// TIA Portal V19 export
FUNCTION_BLOCK "CallInterfaceSignals"   // FB38, LAD
TITLE = CallInterfaceSignals
AUTHOR : Siemens Digital Industry
VERSION : 1.0
// The block serves as a calling interface of the block “LAF_InterfaceSignalsBool“. The block is designed as function block in order to implement the block calls as multi-instances.
// Der Baustein dient als Aufrufschnittstelle für den Funktionsbaustein „LSicar_InterfaceSignalsBool“. Er ist als Funktionsbaustein ausgeführt, um die intern aufgerufenen FBs mittels Multiinstanzen realisieren zu können.  
// Die Funktionsbausteine und das zugehörige WinCC-Bild sind für 16 Signaldatensätze („Schnittstelle Signale 01“ … „Schnittstellen Signale 16“) mit jeweils 32 boolschen Signalen vorgesehen.  
// 
// **PLC-Datentypen**  
//  LSicar_typeInterfaceSignalsBool 
//  typeInterfaceSignalsHmi 
//  LSicar _typeInterfaceSignals 
// 
// **WinCC-Diagnosebild**  
// 
// ![Icon](_Icon/reference.PNG)
// 
// siehe ..\Library Types\LSicar_InterfaceSignalsBool.pdf  
// 
//  
// 
// **Beispielaufruf**  
// Abbildung in Kontaktplan (KOP).  D:\Software\Symbols_Icons\BMPs-JPGs-PNGs\Verschiedene\symb_user_goto_transparent.pngEin lauffähiger Programm-Aufruf hierzu ist im „SICAR-StartUp“-Projekt enthalten.  
// 
// **Aufrufschnittstelle**  
// Der Baustein wird einmalig im zyklischen Programm aufgerufen.  
// 
// **Intern verwendete „Erweiterte Anweisungen / Bausteine“**  
// ..\Library Types\LSicar_InterfaceSignalsBool.pdf
// stored: IsIECCheckEnabled true, MemoryReserve 100, SetENOAutomatically true
   VAR
      statReadValueHmi : Bool;   // HMI: Lese Signalwert / HMI: Read value signal
      statSelectSignalsHmi : USInt := 1;   // HMI: Angewählte Interface Schnittstelle (1..16) / HMI: Selected interface signals (1..16)
      statSelectSignalsOld { ExternalAccessible := 'False'; ExternalVisible := 'False'; ExternalWritable := 'False'} : USInt;   // Altwert: Angewählte Interface Schnittstelle / Old value: Selected interface signals
      statRisEdgeReadName { ExternalAccessible := 'False'; ExternalVisible := 'False'; ExternalWritable := 'False'} : Bool;   // Steigende Flanke / Rising edge
      statPosPulseReadName : Bool;   // Positiver Impuls / Positive pulse
      statInterfaceSignalsHmi : Array[0..16] of "LAF_typeInterfaceSignalsHmi";   // HMI: Beschreibung, Wert und Symbolischer Name / HMI: Description, value and symbolic name
      instSignals1Left { S7_SetPoint := 'True'} : "LAF_InterfaceSignalsBool";
      instSignals1Right { ExternalAccessible := 'False'; ExternalVisible := 'False'; ExternalWritable := 'False'} : "LAF_InterfaceSignalsBool";   // Schnittstellen Signale Bild 1 rechts / interface signals screen 1 right
      instSignals2Left { ExternalAccessible := 'False'; ExternalVisible := 'False'; ExternalWritable := 'False'} : "LAF_InterfaceSignalsBool";   // Schnittstellen Signale Bild 2 links / interface signals screen 2 left
      instSignals2Right { ExternalAccessible := 'False'; ExternalVisible := 'False'; ExternalWritable := 'False'} : "LAF_InterfaceSignalsBool";   // Schnittstellen Signale Bild 2 rechts / interface signals screen 2 right
      instSignals3Left { ExternalAccessible := 'False'; ExternalVisible := 'False'; ExternalWritable := 'False'} : "LAF_InterfaceSignalsBool";   // Schnittstellen Signale Bild 3 links / interface signals screen 3 left
      instSignals3Right { ExternalAccessible := 'False'; ExternalVisible := 'False'; ExternalWritable := 'False'} : "LAF_InterfaceSignalsBool";   // Schnittstellen Signale Bild 3 rechts / interface signals screen 3 right
      instSignals4Left { ExternalAccessible := 'False'; ExternalVisible := 'False'; ExternalWritable := 'False'} : "LAF_InterfaceSignalsBool";   // Schnittstellen Signale Bild 4 links / interface signals screen 4 left
      instSignals4Right { ExternalAccessible := 'False'; ExternalVisible := 'False'; ExternalWritable := 'False'} : "LAF_InterfaceSignalsBool";   // Schnittstellen Signale Bild 4 rechts / interface signals screen 4 right
      instSignals5Left { ExternalAccessible := 'False'; ExternalVisible := 'False'; ExternalWritable := 'False'} : "LAF_InterfaceSignalsBool";   // Schnittstellen Signale Bild 5 links / interface signals screen 5 left
      instSignals5Right { ExternalAccessible := 'False'; ExternalVisible := 'False'; ExternalWritable := 'False'} : "LAF_InterfaceSignalsBool";   // interface signals screen 5 right / Schnittstellen Signale Bild 5 rechts
   END_VAR
   VAR_TEMP
      tempLoopCounter : DInt;   // temp. Schleifenzähler / temp. Loop Counter
   END_VAR
   VAR_TEMP   // added for the SCL form of the ladder/FBD networks
      _w1 : Bool;
   END_VAR
BEGIN

REGION Network 1: BLOCK INFO HEADER / Beschreibung
   // SIEMENS AG / (c)Copyright 2024
   // ------------------------------------------------------------------------------
   // Title:            CallInterfaceSignals (FB38)
   // Comment/Function: The block serves as a calling interface of the block “LAF_InterfaceSignalsBool“. The block is designed as function block in order to implement the block calls as multi-instances. 
   // Library/Family:   -
   // Author:           Siemens Digital Industry
   // Tested with:      ---
   // Engineering:      TIA Portal V19
   // Restrictions:     -
   // Requirements:     ---
   // ------------------------------------------------------------------------------
   // Change log table:
   // Version  | Date       | Expert in charge       | Changes applied
   // ---------|------------|------------------------|------------------------------
   // 01.00.00 | 11.12.2023 | SIMATIC Systems Support 
   //                         First released version
   // **Betriebsart Automatik / Hand**  
   // Der Baustein ist keiner Betriebsart / Betriebsartenbereich zugeordnet.  
   // 
   // **Alarme**  
   // Der Baustein generiert keine Alarme.  
   // 
   // #### PLC-Datentypen  
   // Verwendete PLC-Datentypen für den SPS-Programmbaustein und das zugehörige WinCC-Bild.  
   // 
   // {.pageWidth}
   // ![Image](CallInterfaceSignals/de/image1.PNG)
   //  
   //  
   // #### Bausteinaufrufe 
   // Der Baustein “LSicar_InterfaceSignalsBool“ wird in diesem FB als Multi-Instanz aufgerufen, entspr. nebenstehender beispielhafter Darstellung.  
   // 
   // {.pageWidth}
   // ![Image](CallInterfaceSignals/de/image2.PNG)
   //  
   // Um einen neuen FB aufzurufen, ziehen Sie den FB in ein neues Netzwerk, wählen Sie „Multiinstanz“ aus, vergeben Sie einen Namen und parametrieren Sie den FB-Aufruf.  
   // 
   // {.pageWidth}
   // ![Image](CallInterfaceSignals/de/image3.PNG)
   //  
   //  
   // #### Weitere Hinweise 
   // 
   // #### Updateinfo 
   // 
   // #### Weitere Dokumente 
   // 
   // ![Icon](_Icon/reference.PNG)
   // 
   // ..\Library Types\LSicar_InterfaceSignalsBool.pdf
END_REGION

REGION Network 2: DESCRIPTION
   // Function block and corresponding WinCC screen are prepared for 16 data sets (“InterfaceSignals01“ through .”InterfaceSignals16“) with 32 Boolean signals each.  
   // 
   // **PLC-Data types**   
   // 
   // * LAF_typeInterfaceSignalsBool 
   // * LAF _typeInterfaceSignals 
   // * typeInterfaceSignalsHmi 
   // 
   // **WinCC-Faceplate**  
   // 
   // <None> 
   // 
   // **WinCC Diagnostic screen**   
   // 
   // See: ..\Library Types\LAF_InterfaceSignalsBool.pdf  
   // 
   // **Block call example** 
   // 
   // View in ladder-logic (LAD), without parameter settings.  
   // 
   // 
   // **Calling interface**  
   // 
   // The block is be called once in the cyclic program.  
   // 
   // **Internally used „Extended instructions / blocks“**  
   // 
   // See: ..\Library Types\LAF_InterfaceSignalsBool.pdf
END_REGION

REGION Network 3: Initialization Loop_1 / Initialisierung Loop_1
   // Preset the loop index / Vorbesetzen des Schleifenindex
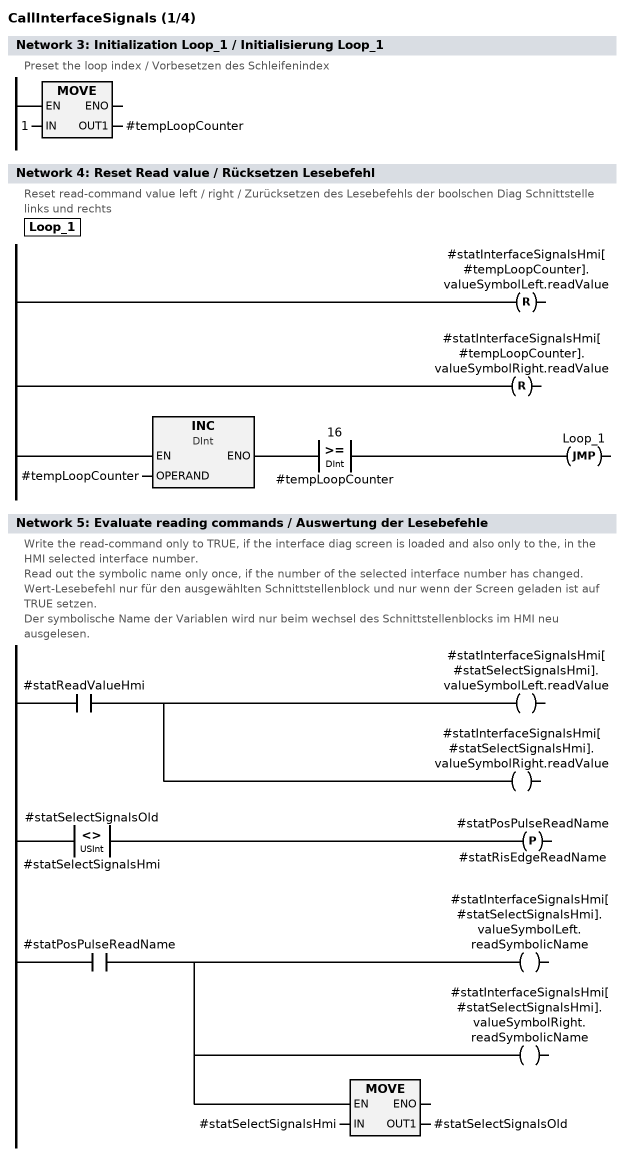
   RUNG wire#powerrail
      Move(in := 1, out1 => #tempLoopCounter)
   END_RUNG
   // the same network as SCL:
   #tempLoopCounter := 1;
END_REGION

REGION Network 4: Reset Read value / Rücksetzen Lesebefehl
   // Reset read-command value left / right / Zurücksetzen des Lesebefehls der boolschen Diag Schnittstelle links und rechts
   Label( Loop_1 )
   RUNG wire#powerrail
      R_Coil( #statInterfaceSignalsHmi[#tempLoopCounter].valueSymbolLeft.readValue )
   END_RUNG
   RUNG wire#powerrail
      R_Coil( #statInterfaceSignalsHmi[#tempLoopCounter].valueSymbolRight.readValue )
   END_RUNG
   RUNG wire#powerrail
      { S7_Templates := "DestType := DInt" } Inc( #tempLoopCounter )
      { S7_Templates := "SrcType := DInt" } GE_Contact(in1 := 16, in2 := #tempLoopCounter)
      JumpCoil( Loop_1 )
   END_RUNG
   // the same network as SCL:
   Loop_1:
   #statInterfaceSignalsHmi[#tempLoopCounter].valueSymbolLeft.readValue := FALSE;
   #statInterfaceSignalsHmi[#tempLoopCounter].valueSymbolRight.readValue := FALSE;
   #tempLoopCounter := #tempLoopCounter + 1;
   IF 16 >= #tempLoopCounter THEN GOTO Loop_1; END_IF;
END_REGION

REGION Network 5: Evaluate reading commands / Auswertung der Lesebefehle
   // Write the read-command only to TRUE, if the interface diag screen is loaded and also only to the, in the HMI selected interface number.
   // Read out the symbolic name only once, if the number of the selected interface number has changed.
   // Wert-Lesebefehl nur für den ausgewählten Schnittstellenblock und nur wenn der Screen geladen ist auf TRUE setzen.
   // Der symbolische Name der Variablen wird nur beim wechsel des Schnittstellenblocks im HMI neu ausgelesen.
   #statInterfaceSignalsHmi[#statSelectSignalsHmi].valueSymbolLeft.readValue := #statReadValueHmi;
   #statInterfaceSignalsHmi[#statSelectSignalsHmi].valueSymbolRight.readValue := #statReadValueHmi;
   #_w1 := #statSelectSignalsOld <> #statSelectSignalsHmi;
   #statPosPulseReadName := #_w1 AND NOT #statRisEdgeReadName;   // rising edge
   #statRisEdgeReadName := #_w1;
   #statInterfaceSignalsHmi[#statSelectSignalsHmi].valueSymbolLeft.readSymbolicName := #statPosPulseReadName;
   #statInterfaceSignalsHmi[#statSelectSignalsHmi].valueSymbolRight.readSymbolicName := #statPosPulseReadName;
   IF #statPosPulseReadName THEN #statSelectSignalsOld := #statSelectSignalsHmi; END_IF;
END_REGION

REGION Network 6: Interface Signals 01 / Interface Signals 01 -Example: Model PosDev+Lifter - IN/OUT-
   // Aufruf des Schnittstellen Signal Bausteins Ba-Bereich 1
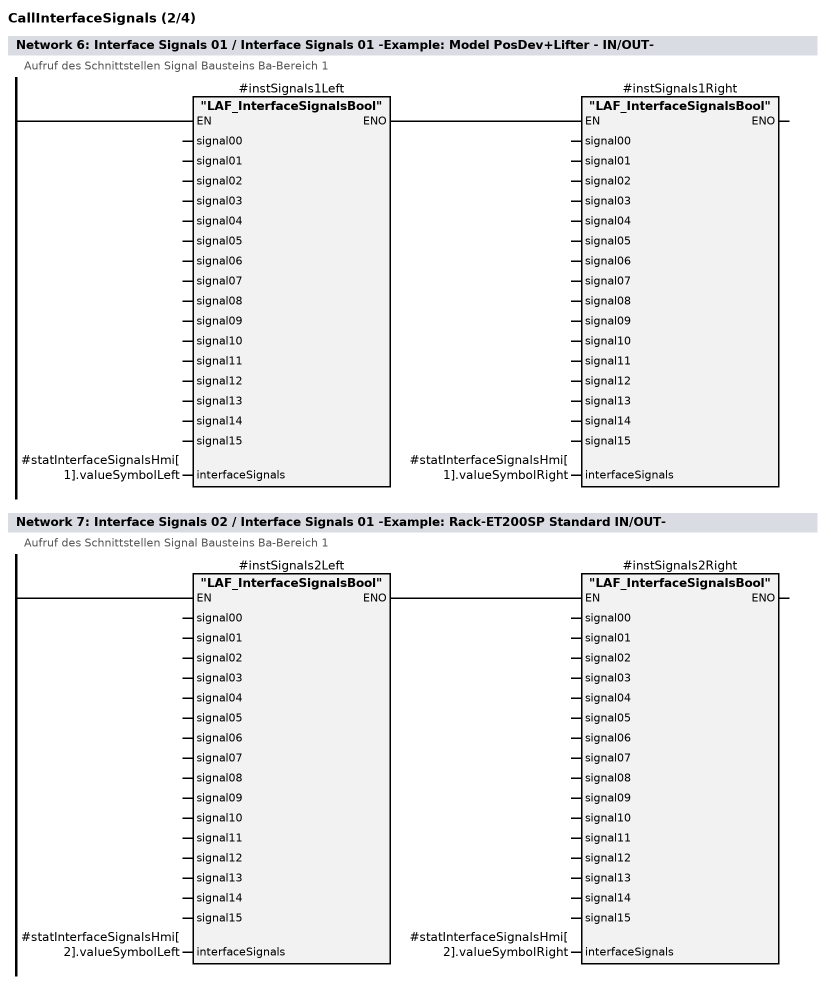
   RUNG wire#powerrail
      #instSignals1Left(signal00 :=, signal01 :=, signal02 :=, signal03 :=, signal04 :=, signal05 :=, signal06 :=, signal07 :=, signal08 :=, signal09 :=, signal10 :=, signal11 :=, signal12 :=, signal13 :=, signal14 :=, signal15 :=, interfaceSignals := #statInterfaceSignalsHmi[1].valueSymbolLeft)
      #instSignals1Right(signal00 :=, signal01 :=, signal02 :=, signal03 :=, signal04 :=, signal05 :=, signal06 :=, signal07 :=, signal08 :=, signal09 :=, signal10 :=, signal11 :=, signal12 :=, signal13 :=, signal14 :=, signal15 :=, interfaceSignals := #statInterfaceSignalsHmi[1].valueSymbolRight)
   END_RUNG
   // the same network as SCL:
   #instSignals1Left(interfaceSignals := #statInterfaceSignalsHmi[1].valueSymbolLeft, ENO => #_w1);   // "LAF_InterfaceSignalsBool"
   IF #_w1 THEN
       #instSignals1Right(interfaceSignals := #statInterfaceSignalsHmi[1].valueSymbolRight);   // "LAF_InterfaceSignalsBool"
   END_IF;
END_REGION

REGION Network 7: Interface Signals 02 / Interface Signals 01 -Example: Rack-ET200SP Standard IN/OUT-
   // Aufruf des Schnittstellen Signal Bausteins Ba-Bereich 1
   RUNG wire#powerrail
      #instSignals2Left(signal00 :=, signal01 :=, signal02 :=, signal03 :=, signal04 :=, signal05 :=, signal06 :=, signal07 :=, signal08 :=, signal09 :=, signal10 :=, signal11 :=, signal12 :=, signal13 :=, signal14 :=, signal15 :=, interfaceSignals := #statInterfaceSignalsHmi[2].valueSymbolLeft)
      #instSignals2Right(signal00 :=, signal01 :=, signal02 :=, signal03 :=, signal04 :=, signal05 :=, signal06 :=, signal07 :=, signal08 :=, signal09 :=, signal10 :=, signal11 :=, signal12 :=, signal13 :=, signal14 :=, signal15 :=, interfaceSignals := #statInterfaceSignalsHmi[2].valueSymbolRight)
   END_RUNG
   // the same network as SCL:
   #instSignals2Left(interfaceSignals := #statInterfaceSignalsHmi[2].valueSymbolLeft, ENO => #_w1);   // "LAF_InterfaceSignalsBool"
   IF #_w1 THEN
       #instSignals2Right(interfaceSignals := #statInterfaceSignalsHmi[2].valueSymbolRight);   // "LAF_InterfaceSignalsBool"
   END_IF;
END_REGION

REGION Network 8: Interface Signals 03 / Interface Signals 03 -Example: System flags & Clock flags-
   // Call the interface signals bool blocks of system tags / Aufruf des Schnittstellen Signal Bausteins für die Systemvariablen
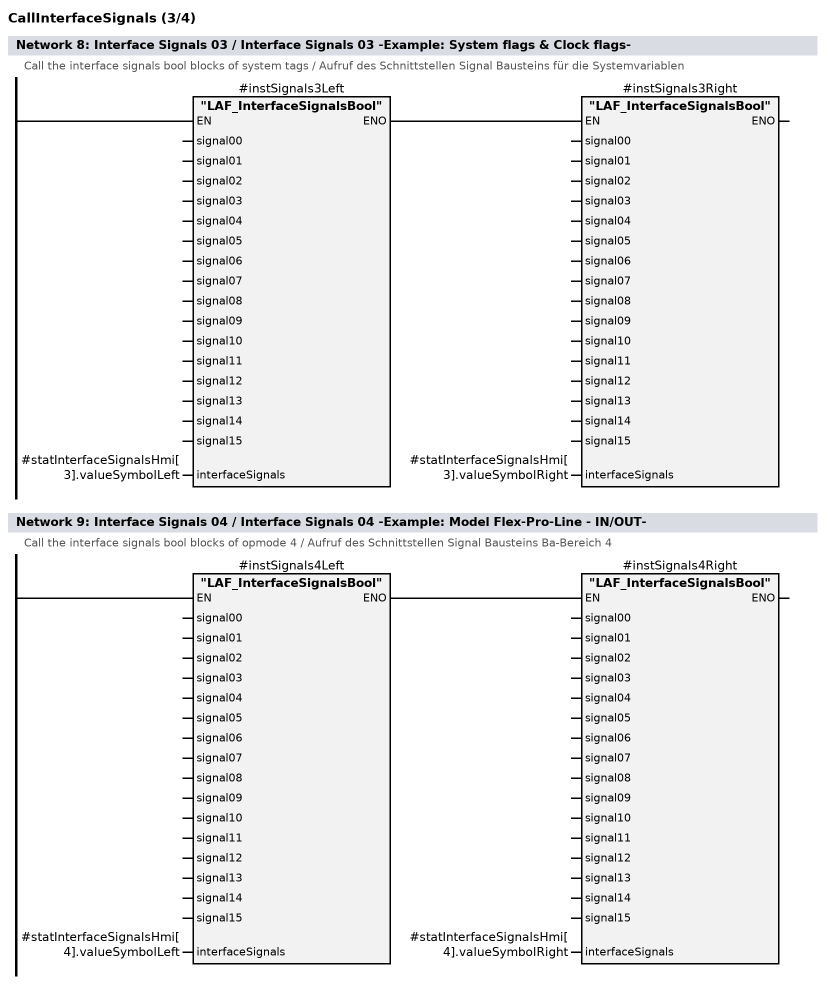
   RUNG wire#powerrail
      #instSignals3Left(signal00 :=, signal01 :=, signal02 :=, signal03 :=, signal04 :=, signal05 :=, signal06 :=, signal07 :=, signal08 :=, signal09 :=, signal10 :=, signal11 :=, signal12 :=, signal13 :=, signal14 :=, signal15 :=, interfaceSignals := #statInterfaceSignalsHmi[3].valueSymbolLeft)
      #instSignals3Right(signal00 :=, signal01 :=, signal02 :=, signal03 :=, signal04 :=, signal05 :=, signal06 :=, signal07 :=, signal08 :=, signal09 :=, signal10 :=, signal11 :=, signal12 :=, signal13 :=, signal14 :=, signal15 :=, interfaceSignals := #statInterfaceSignalsHmi[3].valueSymbolRight)
   END_RUNG
   // the same network as SCL:
   #instSignals3Left(interfaceSignals := #statInterfaceSignalsHmi[3].valueSymbolLeft, ENO => #_w1);   // "LAF_InterfaceSignalsBool"
   IF #_w1 THEN
       #instSignals3Right(interfaceSignals := #statInterfaceSignalsHmi[3].valueSymbolRight);   // "LAF_InterfaceSignalsBool"
   END_IF;
END_REGION

REGION Network 9: Interface Signals 04 / Interface Signals 04 -Example: Model Flex-Pro-Line - IN/OUT-
   // Call the interface signals bool blocks of opmode 4 / Aufruf des Schnittstellen Signal Bausteins Ba-Bereich 4
   RUNG wire#powerrail
      #instSignals4Left(signal00 :=, signal01 :=, signal02 :=, signal03 :=, signal04 :=, signal05 :=, signal06 :=, signal07 :=, signal08 :=, signal09 :=, signal10 :=, signal11 :=, signal12 :=, signal13 :=, signal14 :=, signal15 :=, interfaceSignals := #statInterfaceSignalsHmi[4].valueSymbolLeft)
      #instSignals4Right(signal00 :=, signal01 :=, signal02 :=, signal03 :=, signal04 :=, signal05 :=, signal06 :=, signal07 :=, signal08 :=, signal09 :=, signal10 :=, signal11 :=, signal12 :=, signal13 :=, signal14 :=, signal15 :=, interfaceSignals := #statInterfaceSignalsHmi[4].valueSymbolRight)
   END_RUNG
   // the same network as SCL:
   #instSignals4Left(interfaceSignals := #statInterfaceSignalsHmi[4].valueSymbolLeft, ENO => #_w1);   // "LAF_InterfaceSignalsBool"
   IF #_w1 THEN
       #instSignals4Right(interfaceSignals := #statInterfaceSignalsHmi[4].valueSymbolRight);   // "LAF_InterfaceSignalsBool"
   END_IF;
END_REGION

REGION Network 10: Interface Signals 05 / Interface Signals 05 -Example: Model Flex-Pro-Line - IN/OUT-
   // Call the interface signals bool blocks of opmode 4 / Aufruf des Schnittstellen Signal Bausteins Ba-Bereich 4
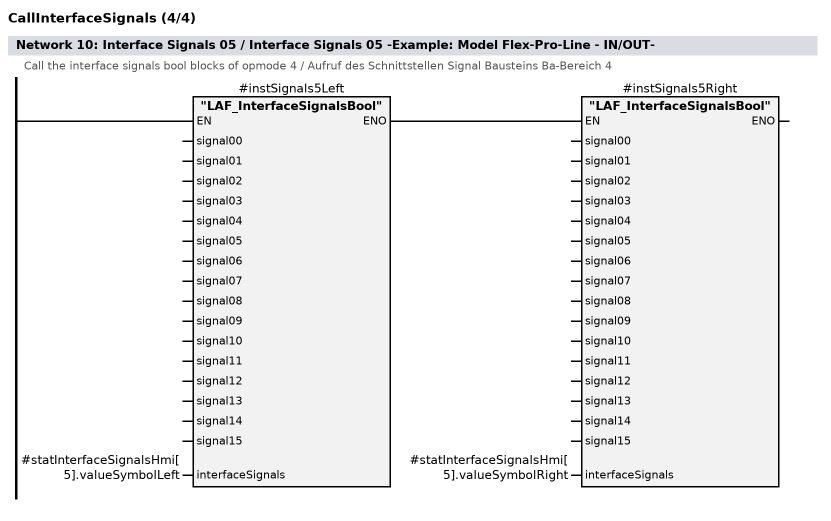
   RUNG wire#powerrail
      #instSignals5Left(signal00 :=, signal01 :=, signal02 :=, signal03 :=, signal04 :=, signal05 :=, signal06 :=, signal07 :=, signal08 :=, signal09 :=, signal10 :=, signal11 :=, signal12 :=, signal13 :=, signal14 :=, signal15 :=, interfaceSignals := #statInterfaceSignalsHmi[5].valueSymbolLeft)
      #instSignals5Right(signal00 :=, signal01 :=, signal02 :=, signal03 :=, signal04 :=, signal05 :=, signal06 :=, signal07 :=, signal08 :=, signal09 :=, signal10 :=, signal11 :=, signal12 :=, signal13 :=, signal14 :=, signal15 :=, interfaceSignals := #statInterfaceSignalsHmi[5].valueSymbolRight)
   END_RUNG
   // the same network as SCL:
   #instSignals5Left(interfaceSignals := #statInterfaceSignalsHmi[5].valueSymbolLeft, ENO => #_w1);   // "LAF_InterfaceSignalsBool"
   IF #_w1 THEN
       #instSignals5Right(interfaceSignals := #statInterfaceSignalsHmi[5].valueSymbolRight);   // "LAF_InterfaceSignalsBool"
   END_IF;
END_REGION

REGION Network 11: Interface Signals 06
   // Call the interface signals bool blocks / Aufruf des Schnittstellen Signal Bausteins
END_REGION

REGION Network 12: Interface Signals 07
   // Call the interface signals bool blocks / Aufruf des Schnittstellen Signal Bausteins
END_REGION

REGION Network 13: Interface Signals 08
   // Call the interface signals bool blocks / Aufruf des Schnittstellen Signal Bausteins
END_REGION

REGION Network 14: Interface Signals 09
   // Call the interface signals bool blocks / Aufruf des Schnittstellen Signal Bausteins
END_REGION

REGION Network 15: Interface Signals 10
   // Call the interface signals bool blocks / Aufruf des Schnittstellen Signal Bausteins
END_REGION

REGION Network 16: Interface Signals 11
   // Call the interface signals bool blocks / Aufruf des Schnittstellen Signal Bausteins
END_REGION

REGION Network 17: Interface Signals 12
   // Call the interface signals bool blocks / Aufruf des Schnittstellen Signal Bausteins
END_REGION

REGION Network 18: Interface Signals 13
   // Call the interface signals bool blocks / Aufruf des Schnittstellen Signal Bausteins
END_REGION

REGION Network 19: Interface Signals 14
   // Call the interface signals bool blocks / Aufruf des Schnittstellen Signal Bausteins
END_REGION

REGION Network 20: Interface Signals 15
   // Call the interface signals bool blocks / Aufruf des Schnittstellen Signal Bausteins
END_REGION

REGION Network 21: Interface Signals 16
   // Call the interface signals bool blocks / Aufruf des Schnittstellen Signal Bausteins
END_REGION
END_FUNCTION_BLOCK
